TYPE ST_Sorter :
{attribute 'OPC.UA.DA' := '1'}
STRUCT
	{attribute 'OPC.UA.DA' := '0'}
	Config				: ST_SorterConfig;
	InductPE			: BOOL;
	EncoderCounts		: UDINT;
	LastUniqueID		: UINT;
	DischargePE			: BOOL;
END_STRUCT
END_TYPE

(* stored: Version 1.1.0.1, ProductVersion 3.1.4024.6
   DUT ST_Sorter: Id {bcb741d2-04a3-4056-8cd7-6667100128c7} *)
